(* IEC 61131-3 sources: plc_generation_empirical_study/datasets/_archive/native_profile_v1_20260810/tasks/C07_M02_temperature_hysteresis, 2 files *)

(* ---- interface.st ---- *)
FUNCTION_BLOCK C07_M02_temperature_hysteresis
VAR_INPUT
    Temperature : REAL;
    LowThreshold : REAL;
    HighThreshold : REAL;
    Enable : BOOL;
END_VAR
VAR_OUTPUT
    Heater : BOOL;
    ConfigError : BOOL;
END_VAR
END_FUNCTION_BLOCK

(* ---- reference.st ---- *)
FUNCTION_BLOCK C07_M02_temperature_hysteresis
VAR_INPUT
    Temperature : REAL;
    LowThreshold : REAL;
    HighThreshold : REAL;
    Enable : BOOL;
END_VAR
VAR_OUTPUT
    Heater : BOOL;
    ConfigError : BOOL;
END_VAR

ConfigError := LowThreshold >= HighThreshold;
IF (NOT Enable) OR ConfigError THEN
    Heater := FALSE;
ELSIF Temperature <= LowThreshold THEN
    Heater := TRUE;
ELSIF Temperature >= HighThreshold THEN
    Heater := FALSE;
END_IF;

END_FUNCTION_BLOCK
